PROGRAM MAIN
VAR
	runOnTime:BOOL:=TRUE; 
END_VAR

IF runOnTime THEN
	ADSLOGSTR(msgCtrlMask:=ADSLOG_MSGTYPE_ERROR OR ADSLOG_MSGTYPE_LOG, msgFmtStr:='Hello %s',strArg:='World');
	runOnTime:=FALSE;
END_IF

END_PROGRAM

(* stored: Version 1.1.0.1, ProductVersion 3.1.4024.9
   POU MAIN: Id {6f278f16-343d-45e9-8f7a-ee2422a7ad6f}, SpecialFunc None *)
